FUNCTION_BLOCK FB_Alive
VAR_INPUT
iAliveSingle:INT;
END_VAR
VAR_OUTPUT
 xQAlive:BOOL;
 xQAliveError:BOOL;
END_VAR
VAR
tTonOff1s:TON;
tTonOn1s:TON;
tTimeOut:ARRAY[1..2] OF TON;
END_VAR

(* 	clock 1 second *)
tTonOff1s(IN:=NOT(tTonOn1s.Q),PT:=t#1s);
tTonOn1s(IN:=(tTonOff1s.Q),PT:=t#1s);

(* Live Bit *)
xQAlive := tTonOff1s.Q;

(*检测是否跳变**)
tTimeOut[1](IN:=(iAliveSingle =1),PT:=T#5S); 
tTimeOut[2](IN:=(iAliveSingle =0),PT:=T#5S); 
xQAliveError:=tTimeOut[1].Q OR tTimeOut[2].Q;

END_FUNCTION_BLOCK

(* stored: Version 1.1.0.1, ProductVersion 3.1.4024.9
   POU FB_Alive: Id {f1f92b40-b4a7-41b1-b839-62ae5064f77c}, SpecialFunc None *)
